TYPE ST_PunchParam :
STRUCT		
	fOverride				: LREAL;
	bCheckPosBeforeRun		: BOOL;
END_STRUCT
END_TYPE

(* stored: Version 1.1.0.1, ProductVersion 3.1.4022.10
   DUT ST_PunchParam: Id {f88b782f-3319-4889-9349-4af439229122} *)
